{attribute 'linkalways'}
{attribute 'no_explicit_call' := 'This FB is a CLASS and must be accessed using methods or properties'}
FUNCTION_BLOCK DefaultAdsLogEventFormatter IMPLEMENTS LogEventFormatter
VAR
END_VAR

METHOD PUBLIC Format : T_MaxString
VAR_INPUT
	event : LogEvent;
END_VAR
VAR_INST
	{attribute 'hide'}
	message_builder : StringBuilder;
END_VAR
VAR CONSTANT
	DELIMITER : STRING := '|';
END_VAR
Format := message_builder
	.Reset()
	.Append(event.logger)
	.Append(DELIMITER)
	.Append(event.message)
	.ToString();
END_METHOD

END_FUNCTION_BLOCK

(* stored: Version 1.1.0.1
   POU DefaultAdsLogEventFormatter: Id {865819e6-2249-459f-9e63-68116177220c}, SpecialFunc None
   Method Format: Id {b32331e9-571d-445c-b5f5-54ca003f258d} *)
